TYPE StationBehaviourInfo :
STRUCT
	MoverId : UDINT;
	CurrentStation : INT;
	Velocity : MC_LREAL;
	State : StationBehaviourState;
END_STRUCT
END_TYPE

(* stored: Version 1.1.0.1
   DUT StationBehaviourInfo: Id {e31e4eaf-6c71-46bd-8e49-86316a781b98} *)
